Fanuc KAREL source: ka00011.KL

PROGRAM KA00011
%NOLOCKGROUP
VAR
SRC:INTEGER
DST : ARRAY[2] OF BYTE
BEGIN
SRC=2
DST[1]=SRC
END KA00011
